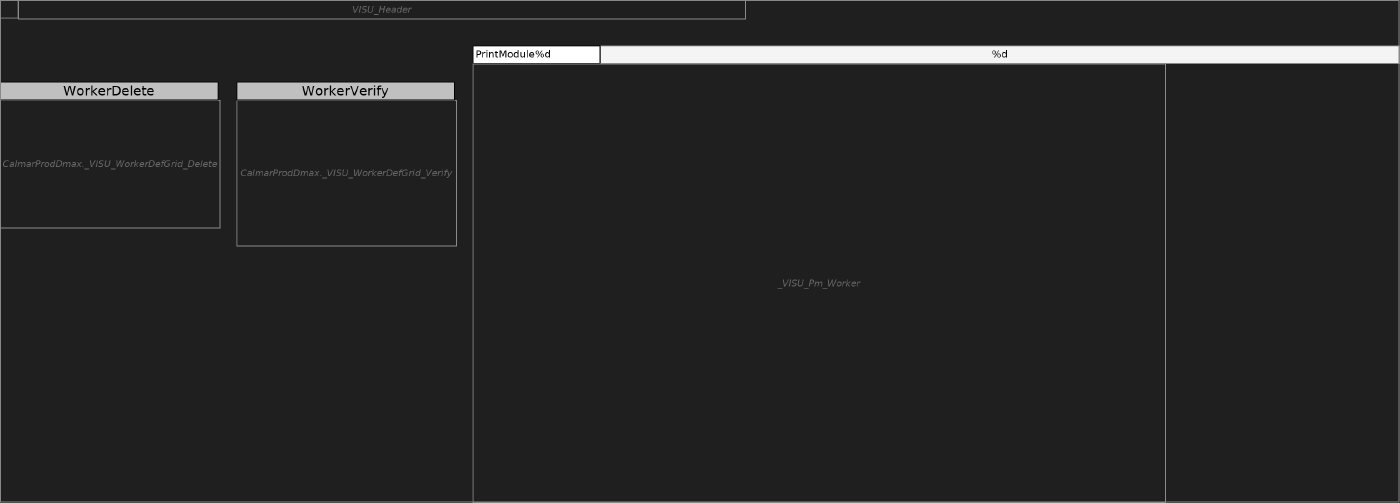
VISUALIZATION VISU_Workers  // 1540x554
    Frame (20,0 800x21)
        shows VISU_Header()
    Scrollbar (660,50 880x20), "%d", text variable: PRG_PRINT.fbModuleMaster.nViewPmSel
        p1057716461: PRG_PRINT.nSelectPmView
    Rectangle (520,50 140x20), "PrintModule%d", text variable: PRG_PRINT.fbModuleMaster.nViewPmSel
    Frame (520,70 762x484)
        shows _VISU_Pm_Worker(mInst := PRG_PRINT.fbPrintModule[PRG_PRINT.fbModuleMaster.nViewPmSel])
    Frame (0,110 242x141)
        shows CalmarProdDmax._VISU_WorkerDefGrid_Delete(m_Inst := PRG_PRINT.fbWorkerDelete)
    Frame (260,110 242x161)
        shows CalmarProdDmax._VISU_WorkerDefGrid_Verify(m_Inst := PRG_PRINT.fbWorkerVerify)
    Rectangle (0,90 240x20), "WorkerDelete"
    Rectangle (260,90 240x20), "WorkerVerify"
    Frame (0,0 20x20)
        shows VISU_ButtonBack()
END_VISUALIZATION

(* stored: Version 1.1.0.1, ProductVersion 3.1.4024.11
   Visu VISU_Workers: Id {4bbef8ba-d0f0-4e80-9afb-448c470105b2} *)
